{attribute addProperty BoxType "EL3214-0000-0016"}
{attribute addProperty Id "RTD_Inputs_ChannelAT %I*ARRAY[0..3] OF RTD_Inputs_Channel_17AE08DB128160WcStateAT %I*WcState_F855686C1620InfoDataAT %I*InfoData_BC63D37F80100"}
{attribute addProperty CRC "449929979"}
{attribute addProperty SizeInBites "224"}
{attribute addProperty SizeInBytes "28"}
TYPE EL3214_6BC1D0AA :
STRUCT
	{attribute addProperty Name "RTD_Inputs_Channel"}
	RTD_Inputs_Channel : ARRAY[0..3] OF RTD_Inputs_Channel_17AE08DB;
	{attribute addProperty Name "WcState"}
	WcState : WcState_F855686C;
	{attribute addProperty Name "InfoData"}
	InfoData : InfoData_BC63D37F;
END_STRUCT
END_TYPE

(* stored: Version 1.2.0.0, ProductVersion 3.1.4024.9
   DUT EL3214_6BC1D0AA: Id {df23ba6f-0ee0-4f9e-9116-2f3b83120999} *)
